FUNCTION_BLOCK StartFeedPositionRot (* Basic Function Block Type *)
  (* Standard: 61499-2 *)
  (* Version 0.0, 7/5/2026, Schneider Electric, Template *)
  PACKAGE SE.Nereda;
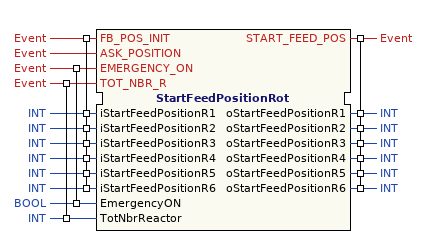
  EVENT_INPUT
    FB_POS_INIT WITH iStartFeedPositionR1, iStartFeedPositionR2, iStartFeedPositionR3, iStartFeedPositionR4, iStartFeedPositionR5, iStartFeedPositionR6;
    ASK_POSITION;
    EMERGENCY_ON WITH EmergencyON;
    TOT_NBR_R WITH TotNbrReactor;
  END_EVENT
  EVENT_OUTPUT
    START_FEED_POS WITH oStartFeedPositionR1, oStartFeedPositionR2, oStartFeedPositionR3, oStartFeedPositionR4, oStartFeedPositionR5, oStartFeedPositionR6;
  END_EVENT
  VAR_INPUT
    iStartFeedPositionR1 : INT;
    iStartFeedPositionR2 : INT;
    iStartFeedPositionR3 : INT;
    iStartFeedPositionR4 : INT;
    iStartFeedPositionR5 : INT;
    iStartFeedPositionR6 : INT;
    EmergencyON : BOOL;
    TotNbrReactor : INT;
  END_VAR
  VAR_OUTPUT
    oStartFeedPositionR1 : INT;
    oStartFeedPositionR2 : INT;
    oStartFeedPositionR3 : INT;
    oStartFeedPositionR4 : INT;
    oStartFeedPositionR5 : INT;
    oStartFeedPositionR6 : INT;
  END_VAR
  VAR
    PositionTab : ARRAY [0..5] OF INT;
    i : INT;
    FirstIndex : INT;
  END_VAR
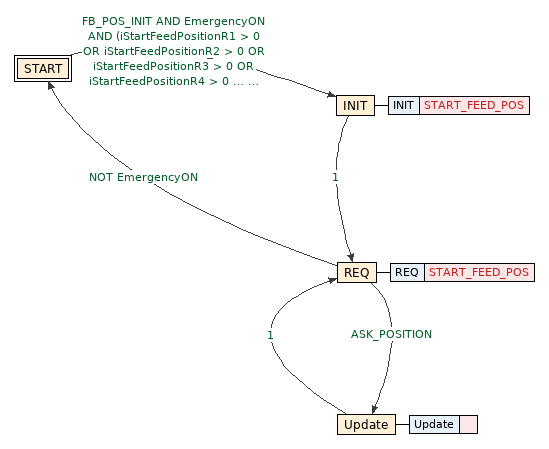
  EC_STATES
    START; (* Initial State *)
    REQ : REQ -> START_FEED_POS; (* Normal execution *)
    INIT : INIT -> START_FEED_POS;
    Update : Update;
  END_STATES
  EC_TRANSITIONS
    START TO INIT := FB_POS_INIT AND EmergencyON AND (iStartFeedPositionR1 > 0 OR iStartFeedPositionR2 > 0 OR iStartFeedPositionR3 > 0 OR iStartFeedPositionR4 > 0 OR iStartFeedPositionR5 > 0 OR iStartFeedPositionR6 > 0);
    REQ TO START := NOT EmergencyON;
    INIT TO REQ := 1;
    REQ TO Update := ASK_POSITION;
    Update TO REQ := 1;
  END_TRANSITIONS
  ALGORITHM REQ IN ST: (* Normally executed algorithm *)
;
FirstIndex := PositionTab[0];
oStartFeedPositionR1 := PositionTab[0];
oStartFeedPositionR2 := PositionTab[1];
oStartFeedPositionR3 := PositionTab[2];
oStartFeedPositionR4 := PositionTab[3];
oStartFeedPositionR5 := PositionTab[4];
oStartFeedPositionR6 := PositionTab[5];
  END_ALGORITHM
  ALGORITHM INIT IN ST:
;
PositionTab[0] := iStartFeedPositionR1;
PositionTab[1] := iStartFeedPositionR2;
PositionTab[2] := iStartFeedPositionR3;
PositionTab[3] := iStartFeedPositionR4;
PositionTab[4] := iStartFeedPositionR5;
PositionTab[5] := iStartFeedPositionR6;
  END_ALGORITHM
  ALGORITHM Update IN ST:
;
IF (TotNbrReactor >= 2) AND (TotNbrReactor <= 6) THEN

    FOR i := 0 TO TotNbrReactor - 2 DO
        PositionTab[i] := PositionTab[i + 1];
    END_FOR;

    PositionTab[TotNbrReactor - 1] := FirstIndex;
END_IF;
  END_ALGORITHM
END_FUNCTION_BLOCK
